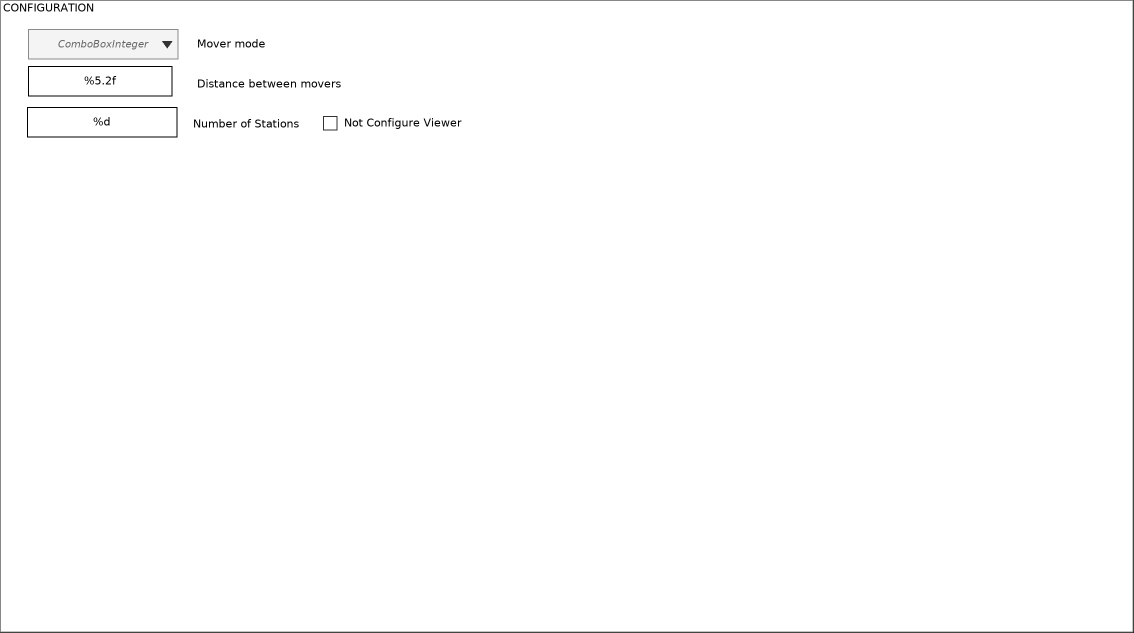
VISUALIZATION VI_XTSConfigurationVisu  // 1134x633
VAR_IN_OUT
	xts : XTS_System;
END_VAR
VAR
	stTableStruct : ARRAY [1..25] OF stTableStructx10;
END_VAR
    Rectangle (0,0 1134x633), "CONFIGURATION"
    Rectangle (27,107 150x30), "%d", text variable: xts.stCfg.udiNumStations
        OnMouseClick: write the text variable via Default
    Label (190,109 150x30), "Number of Stations"
    Checkbox (321,108 165x30), "Not Configure Viewer", variable: xts.stCfg.bNotCfgStationsViewer
    Label (194,29 150x30), "Mover mode"
    ComboBoxInteger (28,29 150x30), variable: xts.stCfg.udiMoverMode, text list: 'MoverMode_TXT'
    Label (194,69 150x30), "Distance between movers"
    Rectangle (28,66 144x30), "%5.2f", text variable: xts.stCfg.lrMoverDistance
        OnMouseClick: write the text variable via Default
END_VISUALIZATION

(* stored: Version 1.1.0.1, ProductVersion 3.1.4024.11
   Visu VI_XTSConfigurationVisu: Id {063e2089-6a55-47b1-b0c7-c8644bd955c4} *)
